(*

short summary
=============

.. <legal notes>

legal notes
=================
| SPDX-FileCopyrightText: © 2023 ekvip automation GmbH <info@ekvip.de>
| SPDX-License-Identifier: Apache-2.0
| For details check: Apache-2.0_

.. _Apache-2.0: https://www.apache.org/licenses/LICENSE-2.0

.. </legal notes>

*)

{warning 'header is generated please add your documentation'}
INTERFACE IReal EXTENDS CNM_AbstractObject.IObject

(*

short summary
=============

.. <legal notes>

legal notes
=================
| SPDX-FileCopyrightText: © 2023 ekvip automation GmbH <info@ekvip.de>
| SPDX-License-Identifier: Apache-2.0
| For details check: Apache-2.0_

.. _Apache-2.0: https://www.apache.org/licenses/LICENSE-2.0

.. </legal notes>

*)

{warning 'header is generated please add your documentation'}
PROPERTY value : REAL
GET
END_GET
SET
END_SET
END_PROPERTY

END_INTERFACE

(* stored: Version 1.1.0.1, ProductVersion 3.1.4024.12
   Itf IReal: Id {9f4edea2-080e-4e01-a88e-ac3fe07f4d24}
   Property value: Id {6959d8ff-79c4-40a8-9dae-0b2e29fea1f8}
   Get Get: Id {dcb33a07-bd80-4c1b-b54d-8800e26dbab8}
   Set Set: Id {02bea2cb-9718-49e2-86dc-8a290fb3755f} *)
